(* IEC 61131-3 sources: HappyLearnCodesys/content/softmotion/CNC11_CustomFunctions, 4 files *)

(* ---- GVL.st ---- *)
{attribute 'qualified_only'}
VAR_GLOBAL
    g_Sel : CNC_Sel;
	g_longline : BOOL;
END_VAR

(* ---- CNC_Sel.st ---- *)
FUNCTION_BLOCK CNC_Sel IMPLEMENTS SMC_NC_IFunction
VAR
    argTypes : ARRAY[0..2] OF SMC_GVar_Type :=
		[SMC_GVar_Type.T_BOOL,
		 SMC_GVar_Type.T_OTHER,
		 SMC_GVar_Type.T_OTHER];
END_VAR

(* ---- CNC.st ---- *)
PROGRAM CNC
VAR
	iState : INT;
	pX, pY, pZ : MC_Power;

	ipo : SMC_Interpolator;
	trafo : SMC_TRAFO_Gantry3;
	trafof : SMC_TRAFOF_Gantry3D;
	cabpX, cabpY, cabpZ : SMC_ControlAxisByPos;
END_VAR

pX(
	Enable:= TRUE,
	bRegulatorOn:= TRUE,
	bDriveStart:= TRUE,
	Axis:= AxisX);

pY(
	Enable:= TRUE,
	bRegulatorOn:= TRUE,
	bDriveStart:= TRUE,
	Axis:= AxisY);

pZ(
	Enable:= TRUE,
	bRegulatorOn:= TRUE,
	bDriveStart:= TRUE,
	Axis:= AxisZ);

CASE iState OF
0:
	IF pX.Status AND pY.Status AND pZ.Status THEN
		iState := 100;
	END_IF

100:
	Interpolation();
END_CASE

(* ---- CNC_PreparePath.st ---- *)
PROGRAM CNC_PreparePath
VAR_INPUT
	xStart : BOOL;
	sFileName : STRING := 'Application/CNC.cnc';
END_VAR
VAR_OUTPUT
	xStartIpo : BOOL;
	poqPath : POINTER TO SMC_Outqueue;
END_VAR
VAR
	iState : INT;
	rncf2 : SMC_ReadNCFile2 := (bParenthesesAsComments:= FALSE);
	nci : SMC_NCInterpreter;
	cv : SMC_CheckVelocities;
	aBufInterpreter : ARRAY[0..99] OF SMC_GeoInfo;
	gcv : SMC_GCodeViewer;

	bufGCV : ARRAY[0..99] OF SMC_GCODEVIEWER_DATA;

    aCNCFunctions : ARRAY[0..0] OF SMC_NC_GFunction :=
        [(stName:= 'SEL', iFunc:= GVL.g_Sel)];

    funTable : SMC_NC_GFunctionTable :=
        (numFunctions:= 1,
         pFunction:= ADR(aCNCFunctions)) ;

	vars : ARRAY[0..0] OF SMC_SingleVar :=
		[
			(strVarName:= 'LONGLINE',
			 eVarType:= SMC_VARTYPE.SMC_TYPE_BOOL,
			 pAdr:= ADR(GVL.g_longline))
		];

	varList : SMC_VARLIST := (wNumberVars:= 1, psvVarList:= ADR(vars));
END_VAR

poqPath := cv.poqDataOut;

gcv(
	GCodeText:= nci.GCodeText,
	bEnable:= TRUE,
	interpolatedObjectId:= CNC.ipo.actObjectId,
	uiNumberOfBufferEntries:= SIZEOF(bufGCV)/SIZEOF(bufGCV[0]),
	pBuffer:= ADR(bufGCV));

CASE iState OF
0:	// idle
	IF xStart THEN
		xStartIpo := FALSE;
		rncf2(bExecute:= FALSE);
		nci(bExecute:= FALSE, sentences:= rncf2.sentences);
		cv(bExecute:= FALSE);

		xStart:=FALSE;
		iState := 10;
	END_IF

10:	// start reading and processing
	rncf2(
        bExecute:= TRUE,
		sFileName:= sFileName,
        pCustomFunTable:= ADR(funTable),
		pvl:= ADR(varList));

	nci(
        bExecute:= TRUE ,
		sentences:= rncf2.sentences,
		nSizeOutQueue:= SIZEOF(aBufInterpreter) ,
		pbyBufferOutQueue:= ADR(aBufInterpreter));

	cv(
        bExecute:= TRUE,
		poqDataIn:= nci.poqDataOut);

	xStartIpo := TRUE;
	IF NOT cv.bBusy THEN
		iState := 0;
	END_IF
END_CASE
